PROGRAM MAIN
VAR
    _legacyDigitalInspectorTests : LegacyTcoDigitalInspectorTests;
    _digitalInspectorTests       : TcoDigitalInspectorTests;
    _analogueInspectorTests      : TcoAnalogueInspectorTests;
    _dataInspectorTests          : TcoDataInspectorTests;
    _inspectionGroupTests        : TcoInspectionGroupTests;
END_VAR

_legacyDigitalInspectorTests.ProbeRun();
_digitalInspectorTests.ProbeRun();
_analogueInspectorTests.ProbeRun();
_dataInspectorTests.ProbeRun();
_inspectionGroupTests.ProbeRun();

END_PROGRAM

(* stored: Version 1.1.0.1, ProductVersion 3.1.4024.9
   POU MAIN: Id {0e1505e0-974d-0b61-1a31-18a914ff2a51}, SpecialFunc None *)
